// TwinCAT 3 PLC project LightsPLC
// ProgramVersion: 3.1.4023.0
// libraries:
//   Tc2_Standard, * (Beckhoff Automation GmbH)
//   Tc2_System, * (Beckhoff Automation GmbH)
//   Tc3_IotBase, * (Beckhoff Automation GmbH)
//   Tc3_JsonXml, * (Beckhoff Automation GmbH)
//   Tc3_Module, * (Beckhoff Automation GmbH)
// project tree:
//   / PlcTask.TcTTO
//   POUs/ F_Scale.TcPOU, MAIN.TcPOU
// real-time tasks:
//   TASK PlcTask: cycle T#10ms, priority 20, ADS port 350
// I/O:
//   DEVICE Device 1 (EtherCAT) (disabled), AmsNetId 8.53.213.166.2.1
//     Term 1 (EK1200)
// variable links:
//   LightsPLC Instance <-> Device 1 (EtherCAT)/Term 1 (EK1200)/Term 2 (EL1859)
//     PlcTask Inputs/MAIN.bLightSetOn <-> Channel 1/Input
//   LightsPLC Instance <-> Device 1 (EtherCAT)/Term 1 (EK1200)/Term 4 (EL3255)
//     PlcTask Inputs/MAIN.Pot1 <-> AI Standard Channel 1/Value
//     PlcTask Inputs/MAIN.Pot2 <-> AI Standard Channel 2/Value
//   LightsPLC Instance <-> Device 1 (EtherCAT)/Term 1 (EK1200)/Term 5 (EL5151)
//     PlcTask Inputs/MAIN.nLightSetHue <-> ENC Inputs/Counter value

CONFIGURATION LightsPLC
    RESOURCE PLC ON TwinCAT3
        TASK PlcTask(INTERVAL := T#10ms, PRIORITY := 20);
        PROGRAM MAIN WITH PlcTask : MAIN;
    END_RESOURCE
END_CONFIGURATION

// ---- POUs/MAIN.TcPOU
PROGRAM MAIN
VAR
	hueClient:	FB_IotHttpClient := (sHostName := '192.168.1.53', bKeepAlive := TRUE, tConnectionTimeout := T#5S);
	hueRequest:	FB_IotHttpRequest;
	
	jsonParser:	FB_JSONDomParser;
	jsonWriter:	FB_JsonSaxWriter;
	jsonDoc:	SJsonValue;
	jsonLight1:	SJsonValue;
	jsonLight1Status:	SJsonValue;
	jsonLightOn:	SJsonValue;
	jsonLightBrightness:	SJsonValue;
	jsonLightHue:	SJsonValue;
	jsonLightSat:	SJsonValue;
	
	Light1On:	BOOL;
	Light1Brightness:	DINT;
	Light1Hue:	DINT;
	Light1Sat:	DINT;
	
	sContent:	STRING(2048);
	sCommand:	STRING;
	
	bGetLights:	BOOL;
	nState:	INT;
	apiKey:	STRING := 'S9U3UinAsoFCoKTF8iFRW-jewXsCee9qjEFFEYHf';
	tempURI:	STRING;
	
	bLightSetOn	AT %I*:	BOOL;
	nLightSetBri:	INT;
	nLightSetHue	AT %I*:	UINT;
	nLightSetHueAuto:	UDINT;
	nLightSetSat:	INT;
	
	Pot1	AT %I*:	INT;
	Pot2	AT %I*: INT;
	
	Timer:	TON;
	rtSend:	R_TRIG;
	bStep: BOOL;
	bConnected: BOOL;
	bRun: BOOL;
	nErrorCount:	UDINT;
END_VAR

nLightSetBri := F_Scale(Pot1);
nLightSetSat := F_Scale(Pot2);

IF NOT hueClient.bConfigured THEN
	hueClient.nHostPort := 80;
	hueClient.stTLS.bNoServerCertCheck := FALSE;
END_IF

IF bGetLights THEN
	bGetLights := FALSE;
	nState := 10;
END_IF

Timer( IN := NOT Timer.Q, PT := T#100MS);
rtSend(CLK := Timer.Q);

IF hueClient.bConnected THEN
	bConnected := TRUE;
END_IF

CASE nState OF
	0:
		IF (bStep OR bRun) AND hueClient.bConfigured THEN
			bStep := FALSE;
			nState := nState + 1;
		END_IF
		
	1:
		jsonWriter.StartObject();
		jsonWriter.AddKey('on');
		jsonWriter.AddBool(bLightSetOn);
		jsonWriter.AddKey('sat');
		jsonWriter.AddUdint(nLightSetSat);
		jsonWriter.AddKey('bri');
		jsonWriter.AddUdint(nLightSetBri);
		jsonWriter.AddKey('hue');
		jsonWriter.AddUdint(nLightSetHueAuto);
		jsonWriter.EndObject();
		sCommand := jsonWriter.GetDocument();
		jsonWriter.ResetDocument();
		nState := nState + 1;
		
	2:
		tempURI := CONCAT(CONCAT('/api/', apiKey), '/lights/1/state');
		IF hueRequest.SendRequest(sUri := tempURI,
									fbClient := hueClient,
									eRequestType := ETcIotHttpRequestType.HTTP_PUT,
									pContent := ADR(sCommand),
									nContentSize := SIZEOF(sCommand),
									fbHeader := 0) THEN
			nState := nState + 1;
		END_IF
		
	3:
		IF NOT hueRequest.bBusy THEN
			IF hueRequest.bError THEN
				nErrorCount := nErrorCount + 1;
				nState := 1;
			ELSE
				IF (bStep OR bRun) THEN
					bStep := FALSE;
					nState := nState + 1;
				END_IF
			END_IF
		END_IF
		
	4:
		hueClient.Disconnect();
		IF (bStep OR bRun) AND NOT hueClient.bConnected THEN
			bStep := FALSE;
			nState := nState + 1;
		END_IF
		
	5:
		IF (bStep OR bRun) THEN
			bStep := FALSE;
			nState := 0;
		END_IF
		
END_CASE

(*CASE nState OF
	0: //IDLE
		IF rtSend.Q THEN
			nState := nState + 1;
		END_IF
	
	1:
		nLightSetHueAuto := nLightSetHueAuto + 5000;
		IF nLightSetHueAuto = 65000 THEN
			nLightSetHueAuto := 0;
		END_IF
		jsonWriter.StartObject();
		jsonWriter.AddKey('on');
		jsonWriter.AddBool(bLightSetOn);
		jsonWriter.AddKey('sat');
		jsonWriter.AddUdint(nLightSetSat);
		jsonWriter.AddKey('bri');
		jsonWriter.AddUdint(nLightSetBri);
		jsonWriter.AddKey('hue');
		jsonWriter.AddUdint(nLightSetHueAuto);
		jsonWriter.EndObject();
		sCommand := jsonWriter.GetDocument();
		jsonWriter.ResetDocument();
		nState := nState + 1;

	2:
		tempURI := CONCAT(CONCAT('/api/', apiKey), '/lights/1/state');
		IF hueRequest.SendRequest(sUri := tempURI,
									fbClient := hueClient,
									eRequestType := ETcIotHttpRequestType.HTTP_PUT,
									pContent := ADR(sCommand),
									nContentSize := SIZEOF(sCommand),
									fbHeader := 0) THEN
			nState := nState + 1;
		END_IF
		
	3:
		IF NOT hueRequest.bBusy THEN
			IF hueRequest.bError THEN
				nState := 500;
			ELSE
				nState := 10;
			END_IF
		END_IF
	
	10:	//Get Light Status
		tempURI := CONCAT(CONCAT('/api/', apiKey),'/lights');
		IF hueRequest.SendRequest(sUri := tempURI,
								fbClient := hueClient,
								eRequestType := ETciotHttpRequestType.HTTP_GET,
								0, 0, 0) THEN
			nState := nState + 1;
		END_IF
		
	11:
		IF NOT hueRequest.bBusy THEN
			IF hueRequest.bError THEN
				nState := 500;
			ELSE
				hueRequest.GetContent(pContent := ADR(sContent),
										nContentSize := SIZEOF(sContent),
										bSetNullTermination := TRUE);
				IF hueRequest.nStatusCode >= 200 AND hueRequest.nStatusCode < 300 THEN
					jsonDoc := hueRequest.GetJsonDomContent(jsonParser);
					jsonLight1 := jsonParser.FindMember(jsonDoc, '1');
					jsonLight1Status := jsonParser.FindMember(jsonLight1, 'state');
					jsonLightOn := jsonParser.FindMember(jsonLight1Status, 'on');
					jsonLightBrightness := jsonParser.FindMember(jsonLight1Status, 'bri');
					jsonLightHue := jsonParser.FindMember(jsonLight1Status, 'hue');
					jsonLightSat := jsonParser.FindMember(jsonLight1Status, 'sat');
					
					Light1On := jsonParser.GetBool(jsonLightOn);
					Light1Brightness := jsonParser.GetInt(jsonLightBrightness);
					Light1Hue := jsonParser.GetInt(jsonLightHue);
					Light1Sat := jsonParser.GetInt(jsonLightSat);
				END_IF
				nState := 0;
			END_IF
		END_IF
		
END_CASE*)

hueClient.Execute();

END_PROGRAM

// ---- POUs/F_Scale.TcPOU
FUNCTION F_Scale : INT
VAR_INPUT
	Value:	INT;
END_VAR
VAR
END_VAR

F_Scale := TO_INT((255.0/32767.0) * TO_REAL(Value));

END_FUNCTION
